TEXTLIST KProduct
  0 = 'Loading'
  1 = 'Loaded'
  2 = 'Unloading'
  3 = 'Unloaded'
   = ''
END_TEXTLIST

(* stored: Version 1.1.0.1, ProductVersion 3.1.4024.11
   TextList KProduct: Id {920e4342-ffe4-428d-acde-66b4e8b199b2} *)
